INTERFACE ITF_Device

METHOD M_GetState : BOOL
VAR_OUTPUT
	O_stCBMLInfo : stCBMLInfo;
END_VAR
END_METHOD

METHOD M_SetName : BOOL
VAR_INPUT
	sName		: STRING;
END_VAR
END_METHOD

PROPERTY P_stCBMLInfo : stCBMLInfo
GET
END_GET
SET
END_SET
END_PROPERTY

END_INTERFACE

(* stored: Version 1.1.0.1, ProductVersion 3.1.4024.11
   Itf ITF_Device: Id {dca516ab-6f97-406c-abb4-bba53a24c488}
   Method M_GetState: Id {9e652fc5-dda9-49b3-8f28-0dcbe7c88c0e}
   Method M_SetName: Id {7b37e582-63dd-463a-9077-07fc45c4e657}
   Property P_stCBMLInfo: Id {13b97e24-0710-4096-a40f-d4c5bddbdf61}
   Get Get: Id {17b6ff28-acfa-4a46-bc1a-5d5b8e1b19c5}
   Set Set: Id {3dc340ff-434a-432e-a628-bf5b0be5bb6c} *)
